{attribute 'GeneratedUsingTerminal: ER4174-0002-0016'}
{attribute addProperty BoxType "ER4174-0002-0016"}
{attribute addProperty Id "Analog_outputAT %Q*INT2"}
{attribute addProperty CRC "3128867708"}
{attribute addProperty Size "2"}
TYPE AO_Outputs_Channel_BA7EBB7C :
STRUCT
	{attribute addProperty Name "Analog_output"}
	Analog_output AT %Q* : INT;
END_STRUCT
END_TYPE
